FUNCTION ARCSEC_TO_DEG : LREAL
VAR_INPUT
    arcsec : LREAL;
END_VAR
VAR
END_VAR

ARCSEC_TO_DEG := arcsec / 3600.0;

END_FUNCTION

(* stored: Version 1.1.0.1, ProductVersion 3.1.4018.5
   POU ARCSEC_TO_DEG: Id {d61448e5-a157-42c9-8736-33420434d66e}, SpecialFunc None *)
